TYPE STATE:
    STRUCT
        curTime: LREAL;
        dvar_M_p_x AT %Q*: DINT;
        dvar_M_p AT %Q*: enum_E;
        dvar_M_q_y AT %Q*: DINT;
        dvar_M_q_b AT %Q*: BOOL;
    END_STRUCT
END_TYPE

(* stored: ProductVersion 3.1.0.18, Version 1.1.0.1 *)
